FUNCTION_BLOCK EventLogger
VAR
	EventBuffer : ARRAY[1..MAXIMUM_SIZE_OF_EVENT_BUFFER] OF ST_Event;
	EventBufferIndex : INT := 0;
	
	_PersistentEventStorage : I_PersistentEventStorage;
	
END_VAR
VAR CONSTANT
	MAXIMUM_SIZE_OF_EVENT_BUFFER : INT := 100;
END_VAR

(* Returns TRUE if add was succesful, FALSE if buffer is full *)
METHOD PUBLIC AddEvent : BOOL
VAR_INPUT
	eEventType : E_EventType;
	eEventSeverity : TcEventSeverity;
	nEventIdentity : UDINT;
	sEventText : STRING(255);
END_VAR
IF NOT IsEventBufferFull() THEN
	EventBufferIndex := EventBufferIndex + 1;
	EventBuffer[EventBufferIndex].eEventType := eEventType;
	EventBuffer[EventBufferIndex].eEventSeverity := eEventSeverity;
	EventBuffer[EventBufferIndex].nEventIdentity := nEventIdentity;
	EventBuffer[EventBufferIndex].sEventText := sEventText;
	UpdateEventTimestampWithSystemTime(stEvent := EventBuffer[EventBufferIndex]);
	AddEvent := TRUE;
ELSE
	AddEvent := FALSE;
END_IF

_PersistentEventStorage.StoreEvent(stEvent := EventBuffer[EventBufferIndex]);
END_METHOD

METHOD FB_init : BOOL
VAR_INPUT
	bInitRetains : BOOL; // if TRUE, the retain variables are initialized (warm start / cold start)
	bInCopyCode : BOOL;  // if TRUE, the instance afterwards gets moved into the copy code (online change)
	iPersistentEventStorage : I_PersistentEventStorage;
END_VAR
_PersistentEventStorage := iPersistentEventStorage;
END_METHOD

METHOD PUBLIC IsEventBufferFull : BOOL
IF (EventBufferIndex + 1) > MAXIMUM_SIZE_OF_EVENT_BUFFER THEN
	IsEventBufferFull := TRUE;
ELSE
	IsEventBufferFull := FALSE;
END_IF
END_METHOD

END_FUNCTION_BLOCK

(* stored: Version 1.1.0.1, ProductVersion 3.1.4024.12
   POU EventLogger: Id {39ec01bf-a102-4de2-8945-079d53bf9b22}, SpecialFunc None
   Method AddEvent: Id {de359dcb-7c92-4372-817b-5f43b4626823}
   Method FB_init: Id {8892bdda-8c43-472f-9d1b-6cc71b313534}
   Method IsEventBufferFull: Id {22bf5949-16ba-4120-996b-2cfa74aa2bc0} *)
